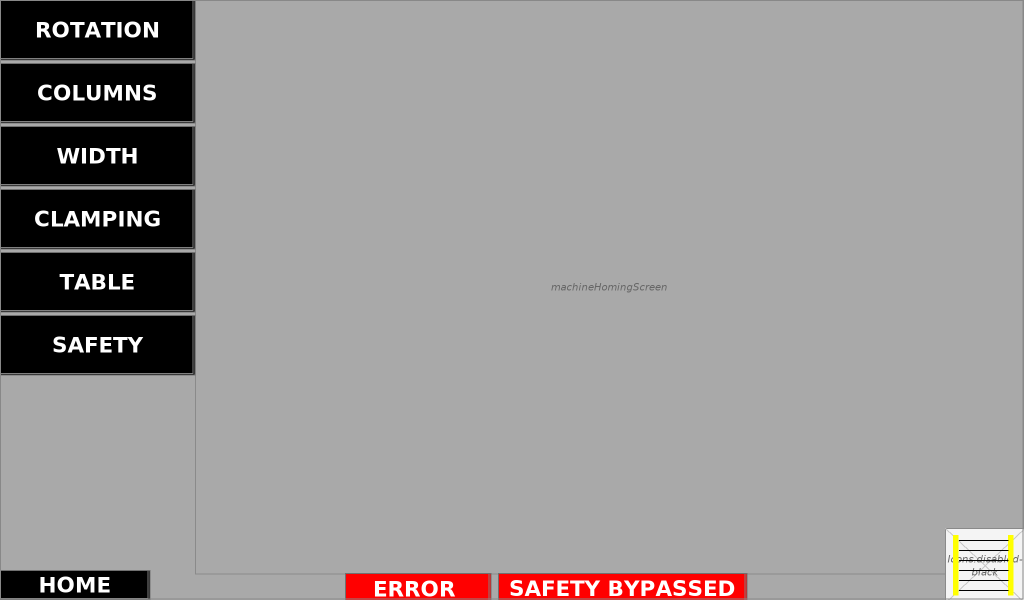
VISUALIZATION maintenance1Screen  // 1024x600
    Button (0,570 150x30), "HOME"
        OnMouseDown: change screen: mainScreen
        OnMouseDown: execute { GVL_machine.nPageIndex := 0; }
    Frame (195,0 829x574), frame switch variable: auto.nFrameDisp
        shows machineHomingScreen()
        shows baseInSkiOutScreen()
        shows loadSpaScreen()
        shows studsInScreen()
        shows unloadSpaScreen()
        shows manualScreen()
        shows safetyResetScreen()
        shows tempEflexScreen()
        shows continueAutoScreen()
    Button (0,0 195x60), "ROTATION"
        toggle auto.bResetBtn
    Button (498,573 249x31), "SAFETY BYPASSED", invisible if: NOT GVL_machine.bSafetyBypass
        OnMouseDown: change screen: safetyDisableWarning
    Button (345,573 146x32), "ERROR", invisible if: NOT GVL_machine.bDispErrorIcon
        OnMouseDown: change screen: errorScreen
    Image (945,528 80x75), invisible if: MAIN.bHideLtCurtainDisable, image: Icons.disabled-black
    Group (953,535 60x60), invisible if: GVL_machine.bSafetyBypass
        toggle GVL_machine.bMuteSafety
        Rectangle (0,0 5x60)
        Rectangle (55,0 5x60)
        Line (6,5) (55,5)
        Line (6,15) (55,15)
        Line (6,25) (55,25)
        Line (6,35) (55,35)
        Line (6,45) (55,45)
        Line (6,55) (55,55)
    Button (0,63 195x60), "COLUMNS"
        toggle auto.bResetBtn
    Button (0,126 195x60), "WIDTH"
        toggle auto.bResetBtn
    Button (0,189 195x60), "CLAMPING"
        toggle auto.bResetBtn
    Button (0,252 195x60), "TABLE"
        toggle auto.bResetBtn
    Button (0,315 195x60), "SAFETY"
        toggle auto.bResetBtn
END_VISUALIZATION

(* stored: Version 1.1.0.1, ProductVersion 3.1.4024.15
   Visu maintenance1Screen: Id {5a80ee74-77aa-42b2-aa02-3bc33f65ce1d} *)
